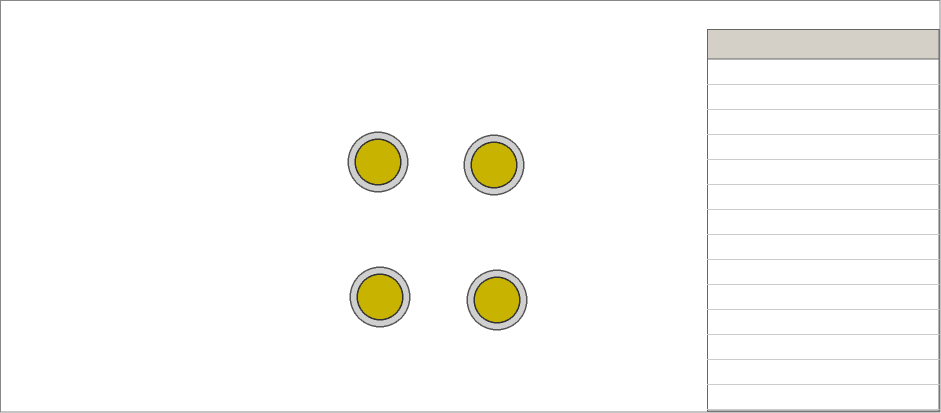
VISUALIZATION Visualization  // 941x413
    Lamp1 (459,130 70x70), variable: MAIN.Switches.str_EnOceanSwitch.bT1_ON, style: Lamp-Lamp1-Yellow
    Lamp1 (345,262 70x70), variable: MAIN.Switches.str_EnOceanSwitch.bT2_ON, style: Lamp-Lamp1-Yellow
    Lamp1 (343,127 70x70), variable: MAIN.Switches.str_EnOceanSwitch.bT1_OFF, style: Lamp-Lamp1-Yellow
    Lamp1 (462,265 70x70), variable: MAIN.Switches.str_EnOceanSwitch.bT2_OFF, style: Lamp-Lamp1-Yellow
    Table (707,29 232x382), data array: MAIN.Search.ar_ID
        p1892666644: MAIN.Search.byNode
        p338671338: MAIN.Search.bReceive
        p2170511999: MAIN.Search.ar_ID
        p3723444502: MAIN.Search.iDevices
        p3854506369: MAIN.Search.ar_ID[INDEX]
END_VISUALIZATION

(* stored: Version 1.1.0.1, ProductVersion 3.1.4022.16
   Visu Visualization: Id {1c4d0898-bfa5-44a9-b2ed-5245603e6a2c} *)
